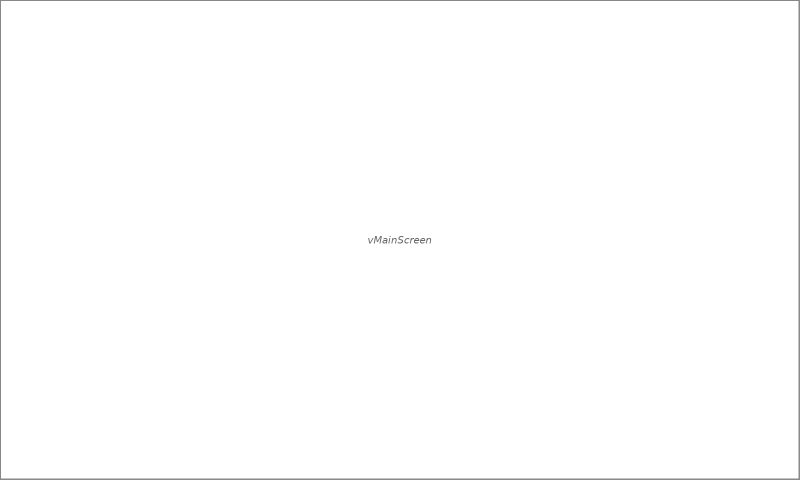
VISUALIZATION vMain  // 800x480
    Frame (0,0 800x480)
        shows vMainScreen(arChamber := MAIN.fb.arFbChamber, arParams := GVL_TesterParams.arstParams, arControl := GVL_TesterParams.arstControl, arTestParams := GVL_TesterParams.arTestParams)
        shows vRecipe(fbChamber := arChamber[iActualChamber], stChamberTestParams := arTestParams[arParams[iActualChamber].iCompresorType])
        shows vService(fbChamber := arChamber[iActualChamber], stParams := arParams[iActualChamber])
        shows vFileSave(fbChamber := arChamber[iActualChamber], stParams := arParams[iActualChamber])
        shows vPlotScreen(stControl := arControl[iActualChamber], fbChamber := arChamber[iActualChamber])
        shows vStatusScreen_v2(arChamber := arChamber[iActualChamber], arParams := arParams[iActualChamber], arControl := arControl[iActualChamber])
END_VISUALIZATION

(* stored: Version 1.1.0.1, ProductVersion 3.1.4024.12
   Visu vMain: Id {ebee01ba-f86c-48f1-94c3-0718742ee16e} *)
